GLOBALCONSTANTS DefaultPool_Numeric (* Numeric object pool constants (ID, Scale, Offset, Decimals) *)
  PACKAGE Uebungen::const::UT::Scroll;
  VAR_GLOBAL CONSTANT
    OutputNumber_12000_N : logiBUS::utils::conversion::phys::NumericObjectPool_S := (u16ObjId := 12000, r32Scale := 1.0, i32Offset := 0, u8Decimals := 0);
    OutputNumber_old_value_N : logiBUS::utils::conversion::phys::NumericObjectPool_S := (u16ObjId := 12001, r32Scale := 0.01, i32Offset := -2147483647, u8Decimals := 2);
    OutputNumber_12002_N : logiBUS::utils::conversion::phys::NumericObjectPool_S := (u16ObjId := 12002, r32Scale := 0.01, i32Offset := -2147483647, u8Decimals := 2);
    OutputNumber_12003_N : logiBUS::utils::conversion::phys::NumericObjectPool_S := (u16ObjId := 12003, r32Scale := 0.01, i32Offset := -2147483647, u8Decimals := 2);
    OutputNumber_new_value_N : logiBUS::utils::conversion::phys::NumericObjectPool_S := (u16ObjId := 12008, r32Scale := 0.01, i32Offset := -2147483647, u8Decimals := 2);
    OutputNumber_Row_03_Value_N : logiBUS::utils::conversion::phys::NumericObjectPool_S := (u16ObjId := 12009, r32Scale := 0.01, i32Offset := -2147483647, u8Decimals := 2);
    OutputNumber_Row_04_Value_N : logiBUS::utils::conversion::phys::NumericObjectPool_S := (u16ObjId := 12010, r32Scale := 0.01, i32Offset := -2147483647, u8Decimals := 2);
    OutputNumber_Row_05_Value_N : logiBUS::utils::conversion::phys::NumericObjectPool_S := (u16ObjId := 12011, r32Scale := 0.01, i32Offset := -2147483647, u8Decimals := 2);
    OutputNumber_Row_06_Value_N : logiBUS::utils::conversion::phys::NumericObjectPool_S := (u16ObjId := 12012, r32Scale := 0.01, i32Offset := -2147483647, u8Decimals := 2);
    OutputNumber_Row_07_Value_N : logiBUS::utils::conversion::phys::NumericObjectPool_S := (u16ObjId := 12013, r32Scale := 0.01, i32Offset := -2147483647, u8Decimals := 2);
    OutputNumber_Row_08_Value_N : logiBUS::utils::conversion::phys::NumericObjectPool_S := (u16ObjId := 12014, r32Scale := 0.01, i32Offset := -2147483647, u8Decimals := 2);
    OutputNumber_Row_09_Value_N : logiBUS::utils::conversion::phys::NumericObjectPool_S := (u16ObjId := 12015, r32Scale := 0.01, i32Offset := -2147483647, u8Decimals := 2);
    OutputNumber_Row_10_Value_N : logiBUS::utils::conversion::phys::NumericObjectPool_S := (u16ObjId := 12016, r32Scale := 0.01, i32Offset := -2147483647, u8Decimals := 2);
    OutputNumber_Row_11_Value_N : logiBUS::utils::conversion::phys::NumericObjectPool_S := (u16ObjId := 12017, r32Scale := 0.01, i32Offset := -2147483647, u8Decimals := 2);
    OutputNumber_Row_12_Value_N : logiBUS::utils::conversion::phys::NumericObjectPool_S := (u16ObjId := 12018, r32Scale := 0.01, i32Offset := -2147483647, u8Decimals := 2);
    OutputNumber_Row_13_Value_N : logiBUS::utils::conversion::phys::NumericObjectPool_S := (u16ObjId := 12019, r32Scale := 0.01, i32Offset := -2147483647, u8Decimals := 2);
    OutputNumber_Row_14_Value_N : logiBUS::utils::conversion::phys::NumericObjectPool_S := (u16ObjId := 12020, r32Scale := 0.01, i32Offset := -2147483647, u8Decimals := 2);
    OutputNumber_Row_15_Value_N : logiBUS::utils::conversion::phys::NumericObjectPool_S := (u16ObjId := 12021, r32Scale := 0.01, i32Offset := -2147483647, u8Decimals := 2);
    OutputNumber_Row_16_Value_N : logiBUS::utils::conversion::phys::NumericObjectPool_S := (u16ObjId := 12022, r32Scale := 0.01, i32Offset := -2147483647, u8Decimals := 2);
    OutputNumber_Row_17_Value_N : logiBUS::utils::conversion::phys::NumericObjectPool_S := (u16ObjId := 12023, r32Scale := 0.01, i32Offset := -2147483647, u8Decimals := 2);
    OutputNumber_Row_18_Value_N : logiBUS::utils::conversion::phys::NumericObjectPool_S := (u16ObjId := 12024, r32Scale := 0.01, i32Offset := -2147483647, u8Decimals := 2);
    OutputNumber_Row_19_Value_N : logiBUS::utils::conversion::phys::NumericObjectPool_S := (u16ObjId := 12025, r32Scale := 0.01, i32Offset := -2147483647, u8Decimals := 2);
    OutputNumber_Row_20_Value_N : logiBUS::utils::conversion::phys::NumericObjectPool_S := (u16ObjId := 12026, r32Scale := 0.01, i32Offset := -2147483647, u8Decimals := 2);
    OutputNumber_Row_03_SubValue_N : logiBUS::utils::conversion::phys::NumericObjectPool_S := (u16ObjId := 12027, r32Scale := 0.01, i32Offset := -2147483647, u8Decimals := 2);
    OutputNumber_Row_04_SubValue_N : logiBUS::utils::conversion::phys::NumericObjectPool_S := (u16ObjId := 12028, r32Scale := 0.01, i32Offset := -2147483647, u8Decimals := 2);
    OutputNumber_Row_05_SubValue_N : logiBUS::utils::conversion::phys::NumericObjectPool_S := (u16ObjId := 12029, r32Scale := 0.01, i32Offset := -2147483647, u8Decimals := 2);
    OutputNumber_Row_06_SubValue_N : logiBUS::utils::conversion::phys::NumericObjectPool_S := (u16ObjId := 12030, r32Scale := 0.01, i32Offset := -2147483647, u8Decimals := 2);
    OutputNumber_Row_07_SubValue_N : logiBUS::utils::conversion::phys::NumericObjectPool_S := (u16ObjId := 12031, r32Scale := 0.01, i32Offset := -2147483647, u8Decimals := 2);
    OutputNumber_Row_08_SubValue_N : logiBUS::utils::conversion::phys::NumericObjectPool_S := (u16ObjId := 12032, r32Scale := 0.01, i32Offset := -2147483647, u8Decimals := 2);
    OutputNumber_Row_09_SubValue_N : logiBUS::utils::conversion::phys::NumericObjectPool_S := (u16ObjId := 12033, r32Scale := 0.01, i32Offset := -2147483647, u8Decimals := 2);
    OutputNumber_Row_10_SubValue_N : logiBUS::utils::conversion::phys::NumericObjectPool_S := (u16ObjId := 12034, r32Scale := 0.01, i32Offset := -2147483647, u8Decimals := 2);
    OutputNumber_Row_11_SubValue_N : logiBUS::utils::conversion::phys::NumericObjectPool_S := (u16ObjId := 12035, r32Scale := 0.01, i32Offset := -2147483647, u8Decimals := 2);
    OutputNumber_Row_12_SubValue_N : logiBUS::utils::conversion::phys::NumericObjectPool_S := (u16ObjId := 12036, r32Scale := 0.01, i32Offset := -2147483647, u8Decimals := 2);
    OutputNumber_Row_13_SubValue_N : logiBUS::utils::conversion::phys::NumericObjectPool_S := (u16ObjId := 12037, r32Scale := 0.01, i32Offset := -2147483647, u8Decimals := 2);
    OutputNumber_Row_14_SubValue_N : logiBUS::utils::conversion::phys::NumericObjectPool_S := (u16ObjId := 12038, r32Scale := 0.01, i32Offset := -2147483647, u8Decimals := 2);
    OutputNumber_Row_15_SubValue_N : logiBUS::utils::conversion::phys::NumericObjectPool_S := (u16ObjId := 12039, r32Scale := 0.01, i32Offset := -2147483647, u8Decimals := 2);
    OutputNumber_Row_16_SubValue_N : logiBUS::utils::conversion::phys::NumericObjectPool_S := (u16ObjId := 12040, r32Scale := 0.01, i32Offset := -2147483647, u8Decimals := 2);
    OutputNumber_Row_17_SubValue_N : logiBUS::utils::conversion::phys::NumericObjectPool_S := (u16ObjId := 12041, r32Scale := 0.01, i32Offset := -2147483647, u8Decimals := 2);
    OutputNumber_Row_18_SubValue_N : logiBUS::utils::conversion::phys::NumericObjectPool_S := (u16ObjId := 12042, r32Scale := 0.01, i32Offset := -2147483647, u8Decimals := 2);
    OutputNumber_Row_19_SubValue_N : logiBUS::utils::conversion::phys::NumericObjectPool_S := (u16ObjId := 12043, r32Scale := 0.01, i32Offset := -2147483647, u8Decimals := 2);
    OutputNumber_Row_20_SubValue_N : logiBUS::utils::conversion::phys::NumericObjectPool_S := (u16ObjId := 12044, r32Scale := 0.01, i32Offset := -2147483647, u8Decimals := 2);
  END_VAR
END_GLOBALCONSTANTS
